Staubli VAL3: Queue.pjx

Parameters version=s7.7.2 stackSize=5000 millimeterUnit=true
Program file=start.pgx
Program file=stop.pgx
Data file=Queue.dtx
Type name=MotionCmd path=../MotionCmd/MotionCmd.pjx
